{attribute 'qualified_only'}
{attribute 'strict'}
TYPE ArmMovementState :
(
	NONE,
	IDLE,
	PICKING,
	DROPPING
);
END_TYPE

(* stored: Version 1.1.0.1, ProductVersion 3.1.4024.12
   DUT ArmMovementState: Id {e3727e3c-51b5-4289-a89b-38cc1bdf6972} *)
